{attribute 'GeneratedUsingTerminal: EL2535-0000-0016'}
{attribute addProperty BoxType "EL2535-0000-0016"}
{attribute addProperty Id "Enable_ditheringBOOL1EnableBOOL1ResetBOOL1"}
{attribute addProperty CRC "625230245"}
{attribute addProperty Size "3"}
TYPE Control_254441A5 :
STRUCT
	{attribute addProperty Name "Enable_dithering"}
	Enable_dithering : BOOL;
	{attribute addProperty Name "Enable"}
	Enable : BOOL;
	{attribute addProperty Name "Reset"}
	Reset : BOOL;
END_STRUCT
END_TYPE

(* stored: Version 1.2.0.0, ProductVersion 3.1.4024.9
   DUT Control_254441A5: Id {b94aa9ed-16f6-40eb-afad-06f94deb0cb3} *)
